// TIA Portal project "S71200Modbus" (V16)

(* hardware
DEVICE "S7-1200 station_1"  S7-1200 Station
   slot 0: "Rack_0"  S7-1200 Rack  Rack  V1.0
   slot 1: "PLC_1"  CPU 1212C AC/DC/Rly  6ES7 212-1BE40-0XB0  V4.4
*)

// ===== PLC "PLC_1"  CPU 1212C AC/DC/Rly =====

VAR_GLOBAL   // PLC tag table "Default tag table"
   "Clock_Byte" AT %MB0 : Byte;
   "Clock_10Hz" AT %M0.0 : Bool;
   "Clock_5Hz" AT %M0.1 : Bool;
   "Clock_2.5Hz" AT %M0.2 : Bool;
   "Clock_2Hz" AT %M0.3 : Bool;
   "Clock_1.25Hz" AT %M0.4 : Bool;
   "Clock_1Hz" AT %M0.5 : Bool;
   "Clock_0.625Hz" AT %M0.6 : Bool;
   "Clock_0.5Hz" AT %M0.7 : Bool;
   "Tag_1" AT %ID100 : DWord;
   "Tag_2" AT %MD5 : UDInt;
   "Tag_3" AT %QD100 : DWord;
   "Tag_4" AT %QD104 : DWord;
   "Tag_5" AT %M10.0 : Bool;
END_VAR

// folder: MBClient

DATA_BLOCK "ClientParameters1"   // DB7
{ S7_Optimized_Access := 'TRUE' }
VERSION : 0.1
   VAR
      Start : Bool;
      Disconnect : Bool;
      Mode : USInt := 0;   // 0:Read; 1:Write
      DataAddress : UDInt := 40001;
      DataLength : UInt := 1;
      Connect : TCON_IP_v4;
      Done : Bool;
      Busy : Bool;
      Error : Bool;
      Status : Word;
   END_VAR
BEGIN
   Connect.InterfaceId := 64;
   Connect.ID := 1;
   Connect.ConnectionType := 11;
   Connect.ActiveEstablished := true;
   Connect.RemoteAddress.ADDR[1] := 192;
   Connect.RemoteAddress.ADDR[2] := 168;
   Connect.RemoteAddress.ADDR[3] := 0;
   Connect.RemoteAddress.ADDR[4] := 70;
   Connect.RemotePort := 14502;
   Connect.LocalPort := 2000;
END_DATA_BLOCK

DATA_BLOCK "DataReceivedH"   // DB8
{ S7_Optimized_Access := 'FALSE' }
VERSION : 0.1
   VAR
      Var : Array[0..15] of Word;
   END_VAR
BEGIN
END_DATA_BLOCK

DATA_BLOCK "MBClient_DB"   // DB9
{ S7_Optimized_Access := 'TRUE' }
VERSION : 0.1
// stored: InstanceOfName MBClient
"MBClient"
BEGIN
END_DATA_BLOCK

DATA_BLOCK "ClientParameters2"   // DB11
{ S7_Optimized_Access := 'TRUE' }
VERSION : 0.1
   VAR
      Disconnect : Bool;
      Mode : USInt := 1;   // 0:Read; 1:Write
      DataAddress : UDInt := 40003;
      DataLength : UInt := 2;
      Connect : TCON_IP_v4;
      Done : Bool;
      Busy : Bool;
      Error : Bool;
      Status : Word;
   END_VAR
BEGIN
   Connect.InterfaceId := 64;
   Connect.ID := 1;
   Connect.ConnectionType := 11;
   Connect.ActiveEstablished := true;
   Connect.RemoteAddress.ADDR[1] := 192;
   Connect.RemoteAddress.ADDR[2] := 168;
   Connect.RemoteAddress.ADDR[3] := 0;
   Connect.RemoteAddress.ADDR[4] := 70;
   Connect.RemotePort := 14502;
   Connect.LocalPort := 2000;
END_DATA_BLOCK

DATA_BLOCK "DataSentH"   // DB12
{ S7_Optimized_Access := 'FALSE' }
VERSION : 0.1
   VAR
      Var : Array[0..15] of Int;
   END_VAR
BEGIN
END_DATA_BLOCK

DATA_BLOCK "DataReceivedB"   // DB15
{ S7_Optimized_Access := 'FALSE' }
VERSION : 0.1
   VAR
      Var : Bool;
   END_VAR
BEGIN
END_DATA_BLOCK

DATA_BLOCK "DataSendB"   // DB16
{ S7_Optimized_Access := 'FALSE' }
VERSION : 0.1
   VAR
      Var : Bool;
   END_VAR
BEGIN
END_DATA_BLOCK

DATA_BLOCK "ClientParameters3"   // DB17
{ S7_Optimized_Access := 'TRUE' }
VERSION : 0.1
   VAR
      Disconnect : Bool;
      Mode : USInt := 0;   // 0:Read; 1:Write
      DataAddress : UDInt := 1;
      DataLength : UInt := 1;
      Connect : TCON_IP_v4;
      Done : Bool;
      Busy : Bool;
      Error : Bool;
      Status : Word;
   END_VAR
BEGIN
   Connect.InterfaceId := 64;
   Connect.ID := 1;
   Connect.ConnectionType := 11;
   Connect.ActiveEstablished := true;
   Connect.RemoteAddress.ADDR[1] := 192;
   Connect.RemoteAddress.ADDR[2] := 168;
   Connect.RemoteAddress.ADDR[3] := 0;
   Connect.RemoteAddress.ADDR[4] := 70;
   Connect.RemotePort := 14502;
   Connect.LocalPort := 2000;
END_DATA_BLOCK

DATA_BLOCK "ClientParameters4"   // DB18
{ S7_Optimized_Access := 'TRUE' }
VERSION : 0.1
   VAR
      Disconnect : Bool;
      Mode : USInt := 1;   // 0:Read; 1:Write
      DataAddress : UDInt := 2;
      DataLength : UInt := 1;
      Connect : TCON_IP_v4;
      Done : Bool;
      Busy : Bool;
      Error : Bool;
      Status : Word;
   END_VAR
BEGIN
   Connect.InterfaceId := 64;
   Connect.ID := 1;
   Connect.ConnectionType := 11;
   Connect.ActiveEstablished := true;
   Connect.RemoteAddress.ADDR[1] := 192;
   Connect.RemoteAddress.ADDR[2] := 168;
   Connect.RemoteAddress.ADDR[3] := 0;
   Connect.RemoteAddress.ADDR[4] := 70;
   Connect.RemotePort := 14502;
   Connect.LocalPort := 2000;
END_DATA_BLOCK

// folder: MBServer

DATA_BLOCK "ServerParameters"   // DB2
{ S7_Optimized_Access := 'TRUE' }
VERSION : 0.1
   VAR
      Disconnect : Bool;
      Connect : TCON_IP_v4;
      NDR : Bool;
      DR : Bool;
      Error : Bool;
      Status : Word;
   END_VAR
BEGIN
   Connect.InterfaceId := 64;
   Connect.ID := 1;
   Connect.ConnectionType := 11;
   Connect.RemoteAddress.ADDR[1] := 0;
   Connect.RemoteAddress.ADDR[2] := 0;
   Connect.RemoteAddress.ADDR[3] := 0;
   Connect.RemoteAddress.ADDR[4] := 0;
   Connect.RemotePort := 0;
   Connect.LocalPort := 502;
END_DATA_BLOCK

DATA_BLOCK "ServerData"   // DB3
{ S7_Optimized_Access := 'FALSE' }
VERSION : 0.1
   VAR
      Var : Array[0..15] of Word;
   END_VAR
BEGIN
END_DATA_BLOCK

DATA_BLOCK "MBServer_DB"   // DB4
{ S7_Optimized_Access := 'TRUE' }
VERSION : 0.1
// stored: InstanceOfName MBServer
"MBServer"
BEGIN
END_DATA_BLOCK

DATA_BLOCK "FactoryData"   // DB5
{ S7_Optimized_Access := 'TRUE' }
VERSION : 0.1
   VAR
      LiquidTempReal : Real;
      LiquidTempDW : DWord;
      FillingTemp : Int;
      DrainingTemp : Int;
   END_VAR
BEGIN
END_DATA_BLOCK

// folder: (top level)

ORGANIZATION_BLOCK "Main"   // OB1, FBD, ProgramCycle
TITLE = "Main Program Sweep (Cycle)"
{ S7_Optimized_Access := 'TRUE' }
VERSION : 0.1
   VAR_INPUT
      Initial_Call : Bool;   // Initial call of this OB
      Remanence : Bool;   // =True, if remanent data are available
   END_VAR
BEGIN

REGION Network 1
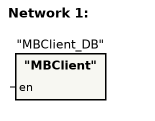
   "MBClient_DB"();   // "MBClient"
END_REGION
END_ORGANIZATION_BLOCK

// folder: MBClient

FUNCTION_BLOCK "MBClient"   // FB2, FBD
{ S7_Optimized_Access := 'TRUE' }
VERSION : 0.1
   VAR_TEMP   // added for the SCL form of the ladder/FBD networks
      _w1 : Bool;
   END_VAR
BEGIN

REGION Network 1: Reading Holding Registers
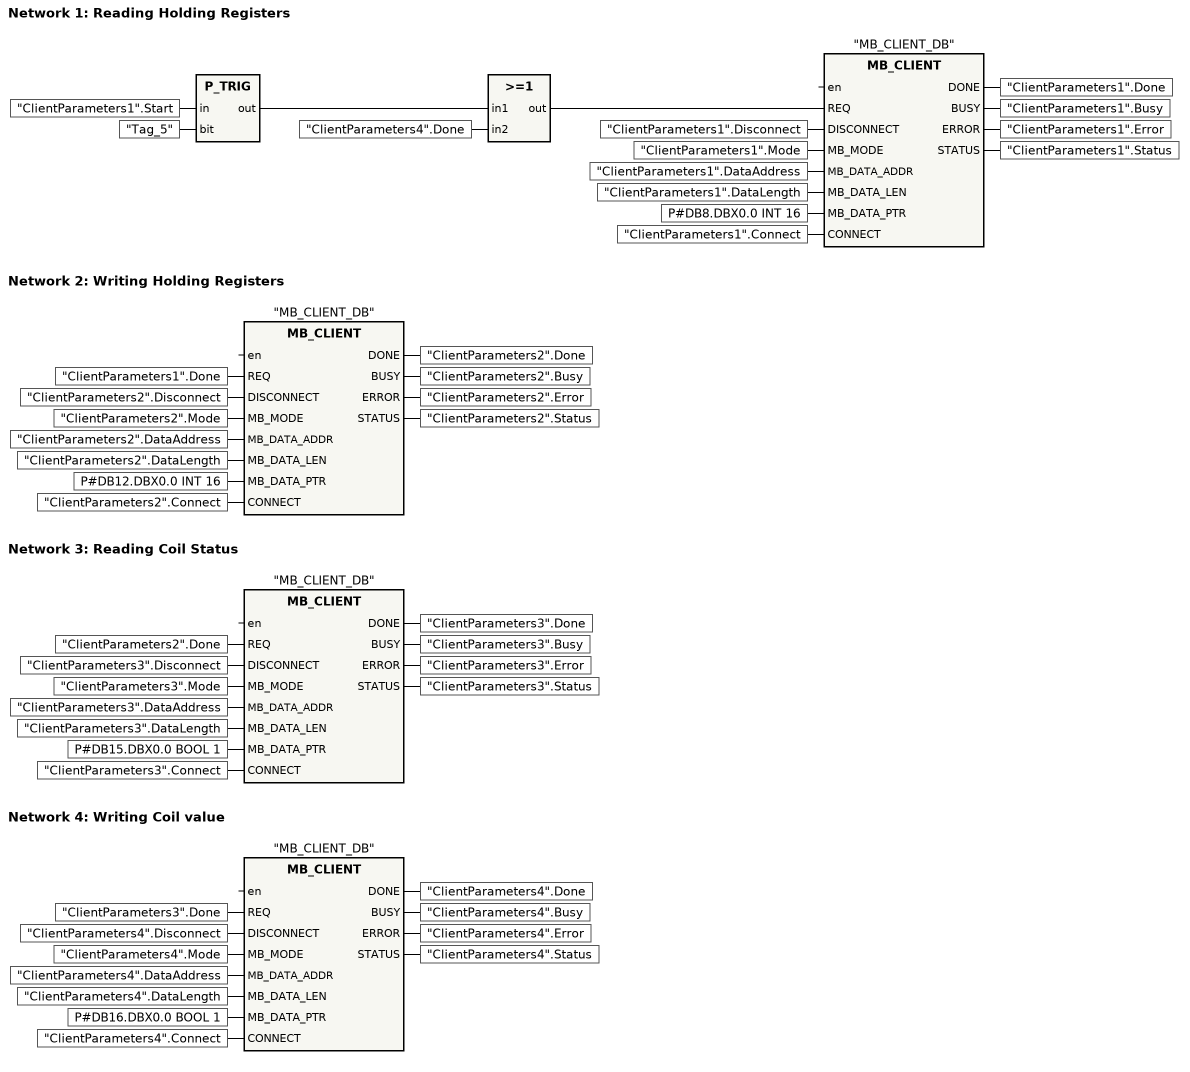
   #_w1 := "ClientParameters1".Start AND NOT "Tag_5";   // rising edge
   "Tag_5" := "ClientParameters1".Start;
   "MB_CLIENT_DB"(REQ := #_w1 OR "ClientParameters4".Done,   // MB_CLIENT
                  DISCONNECT := "ClientParameters1".Disconnect,
                  MB_MODE := "ClientParameters1".Mode,
                  MB_DATA_ADDR := "ClientParameters1".DataAddress,
                  MB_DATA_LEN := "ClientParameters1".DataLength,
                  MB_DATA_PTR := P#DB8.DBX0.0 INT 16,
                  CONNECT := "ClientParameters1".Connect,
                  DONE => "ClientParameters1".Done,
                  BUSY => "ClientParameters1".Busy,
                  ERROR => "ClientParameters1".Error,
                  STATUS => "ClientParameters1".Status);
END_REGION

REGION Network 2: Writing Holding Registers
   "MB_CLIENT_DB"(REQ := "ClientParameters1".Done,   // MB_CLIENT
                  DISCONNECT := "ClientParameters2".Disconnect,
                  MB_MODE := "ClientParameters2".Mode,
                  MB_DATA_ADDR := "ClientParameters2".DataAddress,
                  MB_DATA_LEN := "ClientParameters2".DataLength,
                  MB_DATA_PTR := P#DB12.DBX0.0 INT 16,
                  CONNECT := "ClientParameters2".Connect,
                  DONE => "ClientParameters2".Done,
                  BUSY => "ClientParameters2".Busy,
                  ERROR => "ClientParameters2".Error,
                  STATUS => "ClientParameters2".Status);
END_REGION

REGION Network 3: Reading Coil Status
   "MB_CLIENT_DB"(REQ := "ClientParameters2".Done,   // MB_CLIENT
                  DISCONNECT := "ClientParameters3".Disconnect,
                  MB_MODE := "ClientParameters3".Mode,
                  MB_DATA_ADDR := "ClientParameters3".DataAddress,
                  MB_DATA_LEN := "ClientParameters3".DataLength,
                  MB_DATA_PTR := P#DB15.DBX0.0 BOOL 1,
                  CONNECT := "ClientParameters3".Connect,
                  DONE => "ClientParameters3".Done,
                  BUSY => "ClientParameters3".Busy,
                  ERROR => "ClientParameters3".Error,
                  STATUS => "ClientParameters3".Status);
END_REGION

REGION Network 4: Writing Coil value
   "MB_CLIENT_DB"(REQ := "ClientParameters3".Done,   // MB_CLIENT
                  DISCONNECT := "ClientParameters4".Disconnect,
                  MB_MODE := "ClientParameters4".Mode,
                  MB_DATA_ADDR := "ClientParameters4".DataAddress,
                  MB_DATA_LEN := "ClientParameters4".DataLength,
                  MB_DATA_PTR := P#DB16.DBX0.0 BOOL 1,
                  CONNECT := "ClientParameters4".Connect,
                  DONE => "ClientParameters4".Done,
                  BUSY => "ClientParameters4".Busy,
                  ERROR => "ClientParameters4".Error,
                  STATUS => "ClientParameters4".Status);
END_REGION
END_FUNCTION_BLOCK

// folder: MBServer

FUNCTION_BLOCK "MBServer"   // FB1, FBD
{ S7_Optimized_Access := 'TRUE' }
VERSION : 0.1
BEGIN

REGION Network 1
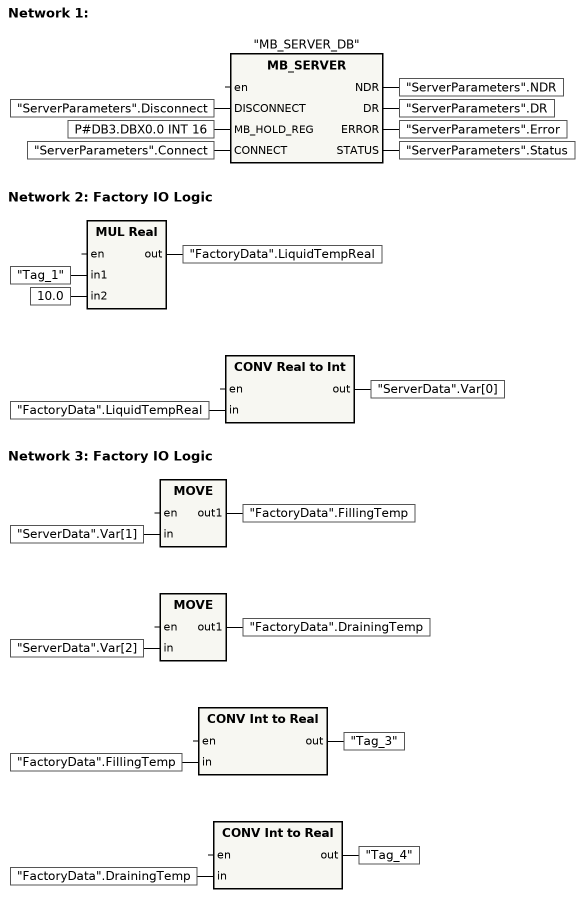
   "MB_SERVER_DB"(DISCONNECT := "ServerParameters".Disconnect,   // MB_SERVER
                  MB_HOLD_REG := P#DB3.DBX0.0 INT 16,
                  CONNECT := "ServerParameters".Connect,
                  NDR => "ServerParameters".NDR,
                  DR => "ServerParameters".DR,
                  ERROR => "ServerParameters".Error,
                  STATUS => "ServerParameters".Status);
END_REGION

REGION Network 2: Factory IO Logic
   // Reading the level
   "FactoryData".LiquidTempReal := "Tag_1" * 10.0;
   "ServerData".Var[0] := REAL_TO_INT("FactoryData".LiquidTempReal);
END_REGION

REGION Network 3: Factory IO Logic
   // Writing the valves
   "FactoryData".FillingTemp := "ServerData".Var[1];
   "FactoryData".DrainingTemp := "ServerData".Var[2];
   "Tag_3" := INT_TO_REAL("FactoryData".FillingTemp);
   "Tag_4" := INT_TO_REAL("FactoryData".DrainingTemp);
END_REGION
END_FUNCTION_BLOCK